{attribute 'GeneratedUsingTerminal: EK1122-0000-0018'}
{attribute addProperty BoxType "EK1122-0000-0018"}
{attribute addProperty Id "Beckhoff_ELXxxxxsub_EK1100EK1100_AB5A94672"}
{attribute addProperty CRC "3521273201"}
{attribute addProperty Size "2"}
TYPE Beckhoff_ELXxxxxEK1122_D1E25D71 EXTENDS EK1122_AB5A9467 :
STRUCT
	{attribute addProperty Name "Beckhoff_ELXxxxxsub_EK1100"}
	Beckhoff_ELXxxxxsub_EK1100 : EK1100_AB5A9467;
END_STRUCT
END_TYPE

(* stored: Version 1.2.0.0, ProductVersion 3.1.4024.9
   DUT Beckhoff_ELXxxxxEK1122_D1E25D71: Id {f775cd6e-6705-4b5b-a9b8-bcc0e74d4581} *)
